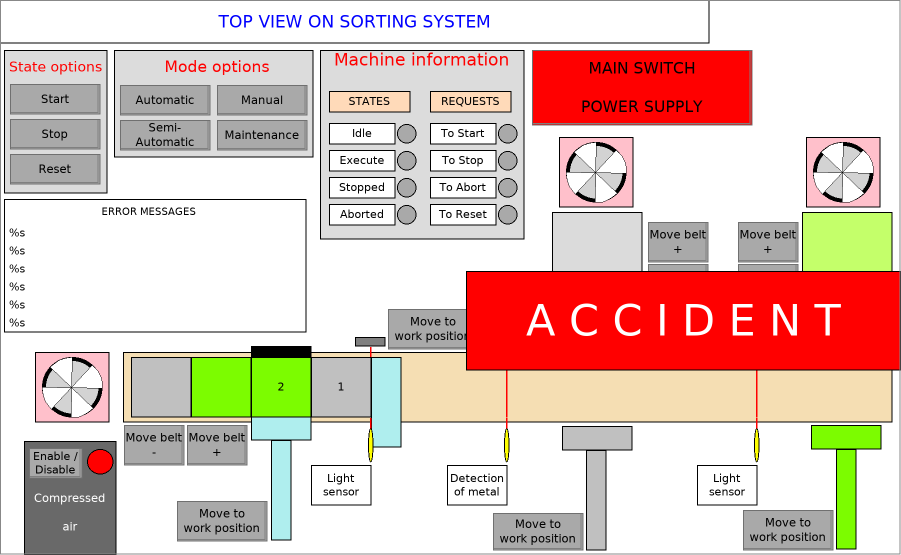
VISUALIZATION Visu_SortingSystem  // 901x555
    Rectangle (123,352 769x70)
    Rectangle (802,212 90x140)
    Rectangle (552,212 90x140)
    Rectangle (741,337 30x9)
    Rectangle (492,337 30x9)
    Ellipse (504,428 5x34)
    Ellipse (754,428 5x34)
    Group (562,426 70x124)
        p2738717112: MAIN.fbMachine.fbVisu.fYMetal
        Rectangle (0,0 70x24)
        Rectangle (24,24 20x100)
    Group (812,426 70x124)
        p2738717112: MAIN.fbMachine.fbVisu.fYPlastic
        Rectangle (-1,-1 70x24)
        Rectangle (24,23 20x100)
    Group (252,417 60x124)
        p2738717112: MAIN.fbMachine.fbVisu.fYClamp
        Rectangle (19,23 20x100)
        Rectangle (-1,-1 60x24)
    Rectangle (131,357 60x60)
        p3560616238: MAIN.fbMachine.fbVisu.aBoxX[4]
        p2738717112: MAIN.fbMachine.fbVisu.aBoxY[4]
    Rectangle (251,357 60x60), "2"
        p3560616238: MAIN.fbMachine.fbVisu.aBoxX[2]
        p2738717112: MAIN.fbMachine.fbVisu.aBoxY[2]
    Rectangle (191,357 60x60)
        p3560616238: MAIN.fbMachine.fbVisu.aBoxX[3]
        p2738717112: MAIN.fbMachine.fbVisu.aBoxY[3]
    Textfield (447,465 60x40), "Detection of metal"
    Textfield (697,465 60x40), "Light sensor"
    Rectangle (506,418 1x10)
    Rectangle (506,347 1x70), invisible if: MAIN.fbMachine.fbMetalSorting.fbSensorDelay.bInput
    Rectangle (756,347 1x70), invisible if: MAIN.fbMachine.fbVisu.bPlasticSensor
    Rectangle (756,418 1x10)
    Textfield (0,0 709x43), "TOP VIEW ON SORTING SYSTEM"
    Rectangle (4,50 103x143)
    Button (10,84 90x30), "Start", colour toggle: MAIN.fbMachine.fbVisu.bButtonColorStart, input disabled if: NOT MAIN.fbMachine.fbVisu.bButtonColorStart AND NOT MAIN.fbMachine.fbVisu.bAccident
        p573394764: MAIN.fbMachine.fbVisu.nButtonColorStart
        toggle MAIN.fbMachine.fbVisu.bButtonStartOut
    Button (10,119 90x30), "Stop", colour toggle: MAIN.fbMachine.fbVisu.bButtonColorStop, input disabled if: NOT MAIN.fbMachine.fbVisu.bButtonColorStop
        p573394764: MAIN.fbMachine.fbVisu.nButtonColorStop
        toggle MAIN.fbMachine.fbVisu.bButtonStopOut
    Button (10,154 90x30), "Reset", colour toggle: MAIN.fbMachine.fbVisu.bButtonColorReset, input disabled if: NOT MAIN.fbMachine.fbVisu.bButtonColorReset
        p573394764: MAIN.fbMachine.fbVisu.nButtonColorReset
        toggle MAIN.fbMachine.fbVisu.bButtonResetOut
    Textfield (7,54 98x25), "State options"
    Rectangle (114,50 199x107)
    Button (120,85 90x30), "Automatic", colour toggle: MAIN.fbMachine.fbVisu.bButtonColorAuto, input disabled if: NOT MAIN.fbMachine.fbVisu.bButtonColorAuto
        p573394764: MAIN.fbMachine.fbVisu.nButtonColorAuto
        toggle MAIN.fbMachine.fbVisu.bButtonAutoOut
    Button (217,85 90x30), "Manual", colour toggle: MAIN.fbMachine.fbVisu.bButtonColorManu, input disabled if: NOT MAIN.fbMachine.fbVisu.bButtonColorManu
        p573394764: MAIN.fbMachine.fbVisu.nButtonColorManu
        toggle MAIN.fbMachine.fbVisu.bButtonManuOut
    Button (120,120 90x30), "Semi- Automatic", colour toggle: MAIN.fbMachine.fbVisu.bButtonColorSemi, input disabled if: NOT MAIN.fbMachine.fbVisu.bButtonColorSemi
        p573394764: MAIN.fbMachine.fbVisu.nButtonColorSemi
        toggle MAIN.fbMachine.fbVisu.bButtonSemiOut
    Button (217,120 90x30), "Maintenance", colour toggle: MAIN.fbMachine.fbVisu.bButtonColorMaint, input disabled if: NOT MAIN.fbMachine.fbVisu.bButtonColorMaint
        p573394764: MAIN.fbMachine.fbVisu.nButtonColorMaint
        toggle MAIN.fbMachine.fbVisu.bButtonMaintenanceOut
    Textfield (156,52 122x29), "Mode options"
    Rectangle (24,441 92x114), "Compressed air"
    Ellipse (87,449 26x25), colour toggle: MAIN.fbMachine.fbVisu.bComprAirEnabled
    Button (648,222 60x40), "Move belt +", colour toggle: MAIN.fbMachine.fbVisu.bButtonColorMetalFw, invisible if: NOT (MAIN.fbMachine.fbVisu.bManual OR MAIN.fbMachine.fbVisu.bMaintenance), input disabled if: NOT MAIN.fbMachine.fbVisu.bButtonColorMetalFw
        p573394764: MAIN.fbMachine.fbVisu.nButtonColorMetalFw
        toggle MAIN.fbMachine.fbVisu.bButtonMetalFwOut
    Button (738,222 60x40), "Move belt +", colour toggle: MAIN.fbMachine.fbVisu.bButtonColorPlasticFw, invisible if: NOT (MAIN.fbMachine.fbVisu.bManual OR MAIN.fbMachine.fbVisu.bMaintenance), input disabled if: NOT MAIN.fbMachine.fbVisu.bButtonColorPlasticFw
        p573394764: MAIN.fbMachine.fbVisu.nButtonColorPlasticFw
        toggle MAIN.fbMachine.fbVisu.bButtonPlasticFwOut
    Button (187,425 60x40), "Move belt +", colour toggle: MAIN.fbMachine.fbVisu.bButtonColorMainFw, invisible if: NOT (MAIN.fbMachine.fbVisu.bManual OR MAIN.fbMachine.fbVisu.bMaintenance), input disabled if: NOT MAIN.fbMachine.fbVisu.bButtonColorMainFw
        p573394764: MAIN.fbMachine.fbVisu.nButtonColorMainFw
        toggle MAIN.fbMachine.fbVisu.bButtonMainFwOut
    Button (648,264 60x40), "Move belt -", colour toggle: MAIN.fbMachine.fbVisu.bButtonColorMetalBw, invisible if: NOT (MAIN.fbMachine.fbVisu.bManual OR MAIN.fbMachine.fbVisu.bMaintenance), input disabled if: NOT MAIN.fbMachine.fbVisu.bButtonColorMetalBw
        p573394764: MAIN.fbMachine.fbVisu.nButtonColorMetalBw
        toggle MAIN.fbMachine.fbVisu.bButtonMetalBwOut
    Button (738,264 60x40), "Move belt -", colour toggle: MAIN.fbMachine.fbVisu.bButtonColorPlasticBw, invisible if: NOT (MAIN.fbMachine.fbVisu.bManual OR MAIN.fbMachine.fbVisu.bMaintenance), input disabled if: NOT MAIN.fbMachine.fbVisu.bButtonColorPlasticBw
        p573394764: MAIN.fbMachine.fbVisu.nButtonColorPlasticBw
        toggle MAIN.fbMachine.fbVisu.bButtonPlasticBwOut
    Button (124,425 60x40), "Move belt -", colour toggle: MAIN.fbMachine.fbVisu.bButtonColorMainBw, invisible if: NOT (MAIN.fbMachine.fbVisu.bManual OR MAIN.fbMachine.fbVisu.bMaintenance), input disabled if: NOT MAIN.fbMachine.fbVisu.bButtonColorMainBw
        p573394764: MAIN.fbMachine.fbVisu.nButtonColorMainBw
        toggle MAIN.fbMachine.fbVisu.bButtonMainBwOut
    Button (388,309 90x40), "Move to work position", colour toggle: MAIN.fbMachine.fbVisu.bButtonColorBarrier, invisible if: NOT (MAIN.fbMachine.fbVisu.bManual OR MAIN.fbMachine.fbVisu.bMaintenance), input disabled if: NOT MAIN.fbMachine.fbVisu.bButtonColorBarrier
        p573394764: MAIN.fbMachine.fbVisu.nButtonColorBarrier
        toggle MAIN.fbMachine.fbVisu.bButtonBarrierToWorkOut
    Button (177,501 90x40), "Move to work position", colour toggle: MAIN.fbMachine.fbVisu.bButtonColorClamp, invisible if: NOT (MAIN.fbMachine.fbVisu.bManual OR MAIN.fbMachine.fbVisu.bMaintenance), input disabled if: NOT MAIN.fbMachine.fbVisu.bButtonColorClamp
        p573394764: MAIN.fbMachine.fbVisu.nButtonColorClamp
        toggle MAIN.fbMachine.fbVisu.bButtonClampToWorkOut
    Button (493,513 90x37), "Move to work position", colour toggle: MAIN.fbMachine.fbVisu.bButtonColorMetalCyl, invisible if: NOT (MAIN.fbMachine.fbVisu.bManual OR MAIN.fbMachine.fbVisu.bMaintenance), input disabled if: NOT MAIN.fbMachine.fbVisu.bButtonColorMetalCyl
        p573394764: MAIN.fbMachine.fbVisu.nButtonColorMetalCyl
        toggle MAIN.fbMachine.fbVisu.bButtonMetalToWorkOut
    Button (743,510 90x40), "Move to work position", colour toggle: MAIN.fbMachine.fbVisu.bButtonColorPlasticCyl, invisible if: NOT (MAIN.fbMachine.fbVisu.bManual OR MAIN.fbMachine.fbVisu.bMaintenance), input disabled if: NOT MAIN.fbMachine.fbVisu.bButtonColorPlasticCyl
        p573394764: MAIN.fbMachine.fbVisu.nButtonColorPlasticCyl
        toggle MAIN.fbMachine.fbVisu.bButtonPlasticToWorkOut
    Rectangle (371,357 30x90)
        p2738717112: MAIN.fbMachine.fbVisu.fYBarrier
    Rectangle (355,337 30x9)
    Ellipse (368,428 5x34)
    Rectangle (370,418 1x10)
    Rectangle (370,347 1x70), invisible if: MAIN.fbMachine.fbVisu.bBarrierSensor
    Textfield (311,465 60x40), "Light sensor"
    Button (532,50 220x75), "MAIN SWITCH POWER SUPPLY", colour toggle: MAIN.fbMachine.fbVisu.bPowerEnabled
        toggle MAIN.fbMachine.fbVisu.bButtonPowerOut
    Rectangle (320,50 204x189), "Machine information"
    Textfield (329,123 66x21), "Idle"
    Textfield (329,150 66x21), "Execute"
    Textfield (329,177 66x21), "Stopped"
    Textfield (329,204 66x21), "Aborted"
    Textfield (430,123 66x21), "To Start"
    Textfield (430,150 66x21), "To Stop"
    Textfield (430,177 66x21), "To Abort"
    Textfield (430,204 66x21), "To Reset"
    Textfield (329,91 81x21), "STATES"
    Textfield (430,91 81x21), "REQUESTS"
    Ellipse (397,124 19x19), colour toggle: MAIN.fbMachine.fbVisu.bIdle
    Ellipse (397,151 19x19), colour toggle: MAIN.fbMachine.fbVisu.bStarted AND MAIN.fbMachine.fbVisu.bPowerEnabled
    Ellipse (397,178 19x19), colour toggle: MAIN.fbMachine.fbVisu.bStopped
    Ellipse (397,205 19x19), colour toggle: MAIN.fbMachine.fbVisu.bAborted
    Ellipse (498,124 19x19), colour toggle: MAIN.fbMachine.fbVisu.bButtonStartIn
    Ellipse (498,151 19x19), colour toggle: MAIN.fbMachine.fbVisu.bButtonStopIn
    Ellipse (498,205 19x19), colour toggle: MAIN.fbMachine.fbVisu.bReset
    Ellipse (498,178 19x19), colour toggle: MAIN.fbMachine.fbVisu.bButtonAbortIn
    Rectangle (251,346 60x11)
    Rectangle (311,357 60x60), "1"
        p3560616238: MAIN.fbMachine.fbVisu.aBoxX[1]
        p2738717112: MAIN.fbMachine.fbVisu.aBoxY[1]
    Button (29,448 53x30), "Enable / Disable", colour toggle: MAIN.fbMachine.fbVisu.bButtonColorComprAir, invisible if: NOT MAIN.fbMachine.fbVisu.bMaintenance, input disabled if: NOT MAIN.fbMachine.fbVisu.bButtonColorComprAir
        p573394764: MAIN.fbMachine.fbVisu.nButtonColorComprAir
        toggle MAIN.fbMachine.fbVisu.bButtonComprAirOut
    Group (4,199 302x133)
        Rectangle (0,0 302x133)
        Textfield (72,3 146x19), "ERROR MESSAGES"
        Textfield (2,26 298x16), "%s", text variable: MAIN.fbMachine.fbVisu.sMessageMainAxis
        Textfield (2,44 298x16), "%s", text variable: MAIN.fbMachine.fbVisu.sMessageMetalAxis
        Textfield (2,62 298x16), "%s", text variable: MAIN.fbMachine.fbVisu.sMessagePlasticAxis
        Textfield (2,80 298x16), "%s", text variable: MAIN.fbMachine.fbVisu.sMessageClamp
        Textfield (2,98 298x16), "%s", text variable: MAIN.fbMachine.fbVisu.sMessageMetalCyl
        Textfield (2,116 298x16), "%s", text variable: MAIN.fbMachine.fbVisu.sMessagePlasticCyl
    Rectangle (466,271 435x99), "A C C I D E N T", invisible if: NOT MAIN.fbMachine.fbVisu.bAccident
    Textfield (35,352 74x70), invisible if: NOT MAIN.fbMachine.fbVisu.bMainAxisMoves
    Rectangle (71,357 1x60)
    Rectangle (42,387 60x1)
    Ellipse (42,357 60x60)
    Polygon (72,357) (71,417) (78,417) (83,415) (88,412) (93,408) (50,367) (47,371) (45,375) (43,380) (42,387) (102,388) (102,382) (101,377) (98,371) (92,365) (51,409) (48,405) (45,401) (43,395) (42,388) (43,382) (44,377) (47,371) (51,366) (55,363) (59,360) (65,358)
        p2858320360: MAIN.fbMachine.fbVisu.nAngleMain
    Textfield (559,137 74x70), invisible if: NOT MAIN.fbMachine.fbVisu.bMetalAxisMoves
    Rectangle (595,142 1x60)
    Rectangle (566,172 60x1)
    Ellipse (566,142 60x60)
    Polygon (596,142) (595,202) (602,202) (607,200) (612,197) (617,193) (574,152) (571,156) (569,160) (567,165) (566,172) (626,173) (626,167) (625,162) (622,156) (616,150) (575,194) (572,190) (569,186) (567,180) (566,173) (567,167) (568,162) (571,156) (575,151) (579,148) (583,145) (589,143)
        p2858320360: MAIN.fbMachine.fbVisu.nAngleMetal
    Textfield (806,137 74x70), invisible if: NOT MAIN.fbMachine.fbVisu.bPlasticAxisMoves
    Rectangle (842,142 1x60)
    Rectangle (813,172 60x1)
    Ellipse (813,142 60x60)
    Polygon (843,142) (842,202) (849,202) (854,200) (859,197) (864,193) (821,152) (818,156) (816,160) (814,165) (813,172) (873,173) (873,167) (872,162) (869,156) (863,150) (822,194) (819,190) (816,186) (814,180) (813,173) (814,167) (815,162) (818,156) (822,151) (826,148) (830,145) (836,143)
        p2858320360: MAIN.fbMachine.fbVisu.nAnglePlastic
END_VISUALIZATION

(* stored: Version 1.1.0.1, ProductVersion 3.1.4024.12
   Visu Visu_SortingSystem: Id {99808b02-9c84-42a4-837f-34ac1c9d7d46} *)
